PROGRAM MAIN
VAR
	Axis1: AXIS_REF;
END_VAR

END_PROGRAM

(* stored: Version 1.1.0.1, ProductVersion 3.1.4024.13
   POU MAIN: Id {f351573f-96fa-47a5-8ea4-1d431a423779}, SpecialFunc None *)
